// TIA Portal V19 export
DATA_BLOCK "Graphics Data"   // DB1
{ S7_Optimized_Access := 'TRUE' }
// stored: MemoryReserve 100
   VAR
      HMI_Graphic_Index : Int;
      HMI_Box_Cnt : DInt;
      HMI_Pallet_Cnt : DInt;
   END_VAR
BEGIN
END_DATA_BLOCK
